FUNCTION Deg_To_Rad : REAL
VAR_INPUT
	fDeg : REAL;
END_VAR
VAR
	fPi : REAL := 3.14159265359;
END_VAR

Deg_To_Rad := (fDeg * fPi)/180;

END_FUNCTION

(* stored: Version 1.1.0.1, ProductVersion 3.1.4024.12
   POU Deg_To_Rad: Id {2368cef4-5365-437d-9566-2947eef801c5}, SpecialFunc None *)
